// TIA Portal V17 export
// export: Created 2022-07-20T06:59:47.1694326Z, ExportSetting WithDefaults, DisplayName Totally Integrated Automation Portal, DisplayVersion V17, DisplayName TIA Portal Openness, DisplayVersion V17, DisplayName TIA Portal Version Control Interface, DisplayVersion V17, DisplayName SINAMICS Startdrive Advanced, DisplayVersion V17, DisplayName SINAMICS Startdrive G130, G150, S120, S150, SINAMICS MV, S210, DisplayVersion V17, DisplayName SINAMICS Startdrive G110M, G120, G120C, G120D, G120P, G115D, DisplayVersion V17, DisplayName STEP 7 Professional, DisplayVersion V17, DisplayName STEP 7 Safety, DisplayVersion V17, DisplayName WinCC Advanced, DisplayVersion V17
FUNCTION_BLOCK "FB10112_OrientalMotorModbusManager"   // FB10112, LAD
TITLE = FB10112_OrientalMotorModbusManager
{ S7_Optimized_Access := 'TRUE' }
AUTHOR : Anirouddh
FAMILY : 1011x_ORIENTAL_MOTOR
VERSION : 1.0
// Release note : 
// 1.0 - Feature developped
// stored: AutoNumber false, IsIECCheckEnabled false, IsRetainMemResEnabled false, MemoryReserve 100, SetENOAutomatically false, UDAEnableTagReadback false
   VAR_INPUT
      MotorInError : Bool;
      OriginPosition : Real;
      WaitingPosition : Real;
      WorkingPosition : Real;
      StepsMmRatio : Real := 500.0;
      RequestAcknowledge : Bool;
      RequestHoming : Bool;
      RequestGoToOriginPosition : Bool;
      RequestGoToWaitingPosition : Bool;
      RequestGoToWorkingPosition : Bool;
      RequestReadActualPosition : Bool;
      RequestReadOriginPosition : Bool;
      RequestReadWaitingPosition : Bool;
      RequestReadWorkingPosition : Bool;
      RequestWriteOriginPosition : Bool;
      RequestWriteWaitingPosition : Bool;
      RequestWriteWorkingPosition : Bool;
      ModbusRequestDone : Bool;
      ModbusDataRegisterToReceive_0 : Int;
      ModbusDataRegisterToReceive_1 : Int;
   END_VAR
   VAR_OUTPUT
      OrientalMotorOutputCommands : "stOrientalModbusStepperMotorCommandOutputs";
      ActualPosition : Real;
      ActualOriginPosition : Real;
      ActualWaitingPosition : Real;
      ActualWorkingPosition : Real;
      HomingDone : Bool;
      IsInOriginPosition : Bool;
      IsInWaitingPosition : Bool;
      IsInWorkingPosition : Bool;
      ReadActualPositionDone : Bool;
      ReadOriginPositionDone : Bool;
      ReadWaitingPositionDone : Bool;
      ReadWorkingPositionDone : Bool;
      ReadAlarmCodeDone : Bool;
      WriteOriginPositionDone : Bool;
      WriteWaitingPositionDone : Bool;
      WriteWorkingPositionDone : Bool;
      StartModbusRtuCommunication : Bool;
      ModbusRtuDataAddress : UInt;
      ModbusRtuDataLength : UInt;
      ModbusRtuMode : USInt;
      ModbusDataRegisterToSend_0 : Int;
      ModbusDataRegisterToSend_1 : Int;
      AlarmStatus : DInt;
      MaterialOK : Bool;
   END_VAR
   VAR
      RequestMotorStartUp : Bool;
      MotorStartUpStateDiagram : Int;
      ModbusCommunicationStateDiagram : Int;
      MotorMovementStateDiagram : Int;
      MotorAlarmManagementStateDiagram : Int;
      ResetStructure : Array[0..31] of Bool;
      R_TRIG_ModbusRequestDone { S7_SetPoint := 'True'} : R_TRIG;
      R_TRIG_RequestHoming { S7_SetPoint := 'True'} : R_TRIG;
      R_TRIG_RequestGoToOriginPosition { S7_SetPoint := 'True'} : R_TRIG;
      R_TRIG_RequestGoToWaitingPosition { S7_SetPoint := 'True'} : R_TRIG;
      R_TRIG_RequestGoToWorkingPosition { S7_SetPoint := 'True'} : R_TRIG;
      R_TRIG_RequestAcknowledge { S7_SetPoint := 'True'} : R_TRIG;
      F_TRIG_MotorInError { S7_SetPoint := 'True'} : F_TRIG;
      TON_HomingSignal { S7_SetPoint := 'True'} : TON_TIME;
      TON_GoToOriginPositionSignal { S7_SetPoint := 'True'} : TON_TIME;
      TON_GoToWaitingPositionSignal { S7_SetPoint := 'True'} : TON_TIME;
      TON_GoToWorkingPositionSignal { S7_SetPoint := 'True'} : TON_TIME;
      TON_AlarmResetSignal { S7_SetPoint := 'True'} : TON_TIME;
   END_VAR
   VAR_TEMP
      ActualPositionTemp : DInt;
      ActualOriginPositionTemp : DInt;
      ActualWaitingPositionTemp : DInt;
      ActualWorkingPositionTemp : DInt;
      ErrorCodeTemp : DInt;
   END_VAR
   VAR CONSTANT
      WAIT_FOR_MOTOR_START_UP : Int := 0;
      INITIALIZE_ORIGIN_POSITION : Int := 10;
      INITIALIZE_WAITING_POSITION : Int := 20;
      INITIALIZE_WORKING_POSITION : Int := 30;
      MOTOR_START_UP_DONE : Int := 40;
      "==========" : Bool;
      WAIT_FOR_MODBUS_COMMUNICATION_REQUEST : Int := 0;
      READ_ACTUAL_POSITION : Int := 10;
      READ_ORIGIN_POSITION : Int := 20;
      READ_WAITING_POSITION : Int := 30;
      READ_WORKING_POSITION : Int := 40;
      WRITE_ORIGIN_POSITION : Int := 50;
      WRITE_WAITING_POSITION : Int := 60;
      WRITE_WORKING_POSITION : Int := 70;
      MODBUS_COMMUNICATION_DONE : Int := 80;
      "==========_1" : Bool;
      WAIT_FOR_MOVEMENT_REQUEST : Int := 0;
      HOMING : Int := 10;
      GO_TO_ORIGIN_POSITION : Int := 20;
      GO_TO_WAITING_POSITION : Int := 30;
      GO_TO_WORKING_POSITION : Int := 40;
      MOVEMENT_DONE : Int := 50;
      "==========_2" : Bool;
      WAIT_FOR_MOTOR_ERROR : Int := 0;
      RESET_MOTOR_COMMUNICATION_MOVEMENT : Int := 10;
      ALARM_RESET : Int := 20;
      GATHER_ERROR_CODE : Int := 30;
      MOTOR_ERROR_MANAGEMENT_DONE : Int := 40;
   END_VAR
BEGIN

REGION Network 1 (SCL): First Scan
   IF "FirstScan" THEN
       #RequestMotorStartUp := TRUE;
       #HomingDone := TRUE;
       #IsInOriginPosition := FALSE;
       #IsInWaitingPosition := FALSE;
       #IsInWorkingPosition := FALSE;
       #ReadActualPositionDone := FALSE;
       #ReadOriginPositionDone := FALSE;
       #ReadWaitingPositionDone := FALSE;
       #ReadWorkingPositionDone := FALSE;
       #ReadAlarmCodeDone := FALSE;
       #WriteOriginPositionDone := FALSE;
       #WriteWaitingPositionDone := FALSE;
       #WriteWorkingPositionDone := FALSE;
       #OrientalMotorOutputCommands.Start := FALSE;
       #OrientalMotorOutputCommands.Stop := FALSE;
       #OrientalMotorOutputCommands.AlarmReset := FALSE;
       #OrientalMotorOutputCommands.M0 := FALSE;
       #OrientalMotorOutputCommands.M1 := FALSE;
       #OrientalMotorOutputCommands.M2 := FALSE;
       #ModbusCommunicationStateDiagram := #WAIT_FOR_MODBUS_COMMUNICATION_REQUEST;
       #MotorMovementStateDiagram := #WAIT_FOR_MOVEMENT_REQUEST;
       #MaterialOK := FALSE;
   END_IF;
END_REGION

REGION Network 2 (SCL): Edge Signals and Timers
   REGION EGDE SIGNALS
       #R_TRIG_ModbusRequestDone(CLK := #ModbusRequestDone AND
                                 (#MotorStartUpStateDiagram = #INITIALIZE_ORIGIN_POSITION OR
                                 #MotorStartUpStateDiagram = #INITIALIZE_WAITING_POSITION OR
                                 #MotorStartUpStateDiagram = #INITIALIZE_WORKING_POSITION));
       #R_TRIG_RequestHoming(CLK := #MotorMovementStateDiagram = #WAIT_FOR_MOVEMENT_REQUEST AND #RequestHoming);
       #R_TRIG_RequestGoToOriginPosition(CLK := #MotorMovementStateDiagram = #WAIT_FOR_MOVEMENT_REQUEST AND #RequestGoToOriginPosition);
       #R_TRIG_RequestGoToWaitingPosition(CLK := #MotorMovementStateDiagram = #WAIT_FOR_MOVEMENT_REQUEST AND #RequestGoToWaitingPosition);
       #R_TRIG_RequestGoToWorkingPosition(CLK := #MotorMovementStateDiagram = #WAIT_FOR_MOVEMENT_REQUEST AND #RequestGoToWorkingPosition);
       #F_TRIG_MotorInError(CLK := #MotorAlarmManagementStateDiagram = #WAIT_FOR_MOTOR_ERROR AND #MotorInError);
       #R_TRIG_RequestAcknowledge(CLK := #MotorAlarmManagementStateDiagram = #WAIT_FOR_MOTOR_ERROR AND #RequestAcknowledge);
   END_REGION


   REGION TIMERS
       //HomingSignal
       #TON_HomingSignal(IN := #MotorMovementStateDiagram = #HOMING,
                         PT := T#15s);

       //GoToOriginPositionSiganl
       #TON_GoToOriginPositionSignal(IN := #MotorMovementStateDiagram = #GO_TO_ORIGIN_POSITION,
                                     PT := T#200ms);

       //GoToWaitingPositionSignal
       #TON_GoToWaitingPositionSignal(IN := #MotorMovementStateDiagram = #GO_TO_WAITING_POSITION,
                                      PT := T#200ms);

       //GoToWorkingPositionSignal
       #TON_GoToWorkingPositionSignal(IN := #MotorMovementStateDiagram = #GO_TO_WORKING_POSITION,
                                      PT := T#200ms);

       //AlarmResetSignal
       #TON_AlarmResetSignal(IN := #MotorAlarmManagementStateDiagram = #ALARM_RESET,
                             PT := T#500ms);
   END_REGION
END_REGION

REGION Network 3 (SCL): Motor Start Up Management
   CASE #MotorStartUpStateDiagram OF
       #WAIT_FOR_MOTOR_START_UP:
           IF #RequestMotorStartUp AND #RequestAcknowledge THEN
               #MotorStartUpStateDiagram := #INITIALIZE_ORIGIN_POSITION;
           END_IF;
       #INITIALIZE_ORIGIN_POSITION:
           #StartModbusRtuCommunication := TRUE;
           #ModbusRtuDataAddress := 41025;
           #ModbusRtuDataLength := 2;
           #ModbusRtuMode := "MODBUS_RTU_WRITE_MODE";
           "FC10332_DWordTo2Words"(DWord_Input := REAL_TO_DINT(#OriginPosition * #StepsMmRatio),
                                Word_HighWeight => #ModbusDataRegisterToSend_0,
                                Word_LowWeight => #ModbusDataRegisterToSend_1);
           IF #R_TRIG_ModbusRequestDone.Q THEN
               #StartModbusRtuCommunication := FALSE;
               #MotorStartUpStateDiagram := #INITIALIZE_WAITING_POSITION;
           END_IF;
       #INITIALIZE_WAITING_POSITION:
           #StartModbusRtuCommunication := TRUE;
           #ModbusRtuDataAddress := 41027;
           #ModbusRtuDataLength := 2;
           #ModbusRtuMode := "MODBUS_RTU_WRITE_MODE";
           "FC10332_DWordTo2Words"(DWord_Input := REAL_TO_DINT(#WaitingPosition * #StepsMmRatio),
                                Word_HighWeight => #ModbusDataRegisterToSend_0,
                                Word_LowWeight => #ModbusDataRegisterToSend_1);
           IF #R_TRIG_ModbusRequestDone.Q THEN
               #StartModbusRtuCommunication := FALSE;
               #MotorStartUpStateDiagram := #INITIALIZE_WORKING_POSITION;
           END_IF;
       #INITIALIZE_WORKING_POSITION:
           #StartModbusRtuCommunication := TRUE;
           #ModbusRtuDataAddress := 40063;
           #ModbusRtuDataLength := 2;
           #ModbusRtuMode := "MODBUS_RTU_WRITE_MODE";
           "FC10332_DWordTo2Words"(DWord_Input := REAL_TO_DINT(#WorkingPosition * #StepsMmRatio),
                                Word_HighWeight => #ModbusDataRegisterToSend_0,
                                Word_LowWeight => #ModbusDataRegisterToSend_1);
           IF #R_TRIG_ModbusRequestDone.Q THEN
               #StartModbusRtuCommunication := FALSE;
               #MotorStartUpStateDiagram := #MOTOR_START_UP_DONE;
           END_IF;
       #MOTOR_START_UP_DONE:
           #MaterialOK := TRUE;
           #RequestMotorStartUp := FALSE;
   END_CASE;
END_REGION

REGION Network 4 (SCL): Modbus Communication Management
   CASE #ModbusCommunicationStateDiagram OF
       #WAIT_FOR_MODBUS_COMMUNICATION_REQUEST:
           IF #RequestReadActualPosition THEN
               #ReadActualPositionDone := FALSE;
               #ReadOriginPositionDone := FALSE;
               #ReadWaitingPositionDone := FALSE;
               #ReadWorkingPositionDone := FALSE;
               #WriteOriginPositionDone := FALSE;
               #WriteWaitingPositionDone := FALSE;
               #WriteWorkingPositionDone := FALSE;
               #ModbusCommunicationStateDiagram := #READ_ACTUAL_POSITION;
           ELSIF #RequestReadOriginPosition THEN
               #ReadActualPositionDone := FALSE;
               #ReadOriginPositionDone := FALSE;
               #ReadWaitingPositionDone := FALSE;
               #ReadWorkingPositionDone := FALSE;
               #WriteOriginPositionDone := FALSE;
               #WriteWaitingPositionDone := FALSE;
               #WriteWorkingPositionDone := FALSE;
               #ModbusCommunicationStateDiagram := #READ_ORIGIN_POSITION;
           ELSIF #RequestReadWaitingPosition THEN
               #ReadActualPositionDone := FALSE;
               #ReadOriginPositionDone := FALSE;
               #ReadWaitingPositionDone := FALSE;
               #ReadWorkingPositionDone := FALSE;
               #WriteOriginPositionDone := FALSE;
               #WriteWaitingPositionDone := FALSE;
               #WriteWorkingPositionDone := FALSE;
               #ModbusCommunicationStateDiagram := #READ_WAITING_POSITION;
           ELSIF #RequestReadWorkingPosition THEN
               #ReadActualPositionDone := FALSE;
               #ReadOriginPositionDone := FALSE;
               #ReadWaitingPositionDone := FALSE;
               #ReadWorkingPositionDone := FALSE;
               #WriteOriginPositionDone := FALSE;
               #WriteWaitingPositionDone := FALSE;
               #WriteWorkingPositionDone := FALSE;
               #ModbusCommunicationStateDiagram := #READ_WORKING_POSITION;
           ELSIF #RequestWriteOriginPosition THEN
               #ReadActualPositionDone := FALSE;
               #ReadOriginPositionDone := FALSE;
               #ReadWaitingPositionDone := FALSE;
               #ReadWorkingPositionDone := FALSE;
               #WriteOriginPositionDone := FALSE;
               #WriteWaitingPositionDone := FALSE;
               #WriteWorkingPositionDone := FALSE;
               #ModbusCommunicationStateDiagram := #WRITE_ORIGIN_POSITION;
           ELSIF #RequestWriteWaitingPosition THEN
               #ReadActualPositionDone := FALSE;
               #ReadOriginPositionDone := FALSE;
               #ReadWaitingPositionDone := FALSE;
               #ReadWorkingPositionDone := FALSE;
               #WriteOriginPositionDone := FALSE;
               #WriteWaitingPositionDone := FALSE;
               #WriteWorkingPositionDone := FALSE;
               #ModbusCommunicationStateDiagram := #WRITE_WAITING_POSITION;
           ELSIF #RequestWriteWorkingPosition THEN
               #ReadActualPositionDone := FALSE;
               #ReadOriginPositionDone := FALSE;
               #ReadWaitingPositionDone := FALSE;
               #ReadWorkingPositionDone := FALSE;
               #WriteOriginPositionDone := FALSE;
               #WriteWaitingPositionDone := FALSE;
               #WriteWorkingPositionDone := FALSE;
               #ModbusCommunicationStateDiagram := #WRITE_WORKING_POSITION;
           END_IF;
       #READ_ACTUAL_POSITION:
           #StartModbusRtuCommunication := TRUE;
           #ModbusRtuDataAddress := 40205;
           #ModbusRtuDataLength := 2;
           #ModbusRtuMode := "MODBUS_RTU_READ_MODE";
           IF #ModbusRequestDone THEN
               "FC10012_2IntToDint"(HighInt := #ModbusDataRegisterToReceive_0,
                                    LowInt := #ModbusDataRegisterToReceive_1,
                                    Output_DInt => #ActualPositionTemp);
               #ActualPosition := DINT_TO_REAL(#ActualPositionTemp) / #StepsMmRatio;
               #ReadActualPositionDone := TRUE;
               #StartModbusRtuCommunication := FALSE;
               #ModbusCommunicationStateDiagram := #MODBUS_COMMUNICATION_DONE;
           END_IF;
       #READ_ORIGIN_POSITION:
           #StartModbusRtuCommunication := TRUE;
           #ModbusRtuDataAddress := 41025;
           #ModbusRtuDataLength := 2;
           #ModbusRtuMode := "MODBUS_RTU_READ_MODE";
           IF #ModbusRequestDone THEN
               "FC10012_2IntToDint"(HighInt := #ModbusDataRegisterToReceive_0,
                                    LowInt := #ModbusDataRegisterToReceive_1,
                                    Output_DInt => #ActualOriginPositionTemp);
               #ActualOriginPosition := DINT_TO_REAL(#ActualOriginPositionTemp) / #StepsMmRatio;
               #ReadOriginPositionDone := TRUE;
               #StartModbusRtuCommunication := FALSE;
               #ModbusCommunicationStateDiagram := #MODBUS_COMMUNICATION_DONE;
           END_IF;
       #READ_WAITING_POSITION:
           #StartModbusRtuCommunication := TRUE;
           #ModbusRtuDataAddress := 41027;
           #ModbusRtuDataLength := 2;
           #ModbusRtuMode := "MODBUS_RTU_READ_MODE";
           IF #ModbusRequestDone THEN
               "FC10012_2IntToDint"(HighInt := #ModbusDataRegisterToReceive_0,
                                    LowInt := #ModbusDataRegisterToReceive_1,
                                    Output_DInt => #ActualWaitingPositionTemp);
               #ActualWaitingPosition := DINT_TO_REAL(#ActualWaitingPositionTemp) / #StepsMmRatio;
               #ReadWaitingPositionDone := TRUE;
               #StartModbusRtuCommunication := FALSE;
               #ModbusCommunicationStateDiagram := #MODBUS_COMMUNICATION_DONE;
           END_IF;
       #READ_WORKING_POSITION:
           #StartModbusRtuCommunication := TRUE;
           #ModbusRtuDataAddress := 41029;
           #ModbusRtuDataLength := 2;
           #ModbusRtuMode := "MODBUS_RTU_READ_MODE";
           IF #ModbusRequestDone THEN
               "FC10012_2IntToDint"(HighInt := #ModbusDataRegisterToReceive_0,
                                    LowInt := #ModbusDataRegisterToReceive_1,
                                    Output_DInt => #ActualWorkingPositionTemp);
               #ActualWorkingPosition := DINT_TO_REAL(#ActualWorkingPositionTemp) / #StepsMmRatio;
               #ReadWorkingPositionDone := TRUE;
               #StartModbusRtuCommunication := FALSE;
               #ModbusCommunicationStateDiagram := #MODBUS_COMMUNICATION_DONE;
           END_IF;
       #WRITE_ORIGIN_POSITION:
           REGION To test later
       (*    #StartModbusRtuCommunication := TRUE;
           #ModbusRtuDataAddress := 44929;
           #ModbusRtuDataLength := 14;
           #ModbusRtuMode := "MODBUS_RTU_WRITE_MODE";
           (*Process Line Update*)
           //Name -> Line Number
           #ModbusDataRegisterToSend[0] := 0;
           #ModbusDataRegisterToSend[1] := 1;
           //Operation Type
           #ModbusDataRegisterToSend[2] := 1; //AbsolutePositionning
           #ModbusDataRegisterToSend[3] := 0;
           //Position
           "FC10011_DintTo2Int"(Dint_Input := REAL_TO_DINT(#OriginPosition * #StepMmRatio),
                                Int_HighWeight => #ModbusDataRegisterToSend[4],
                                Int_LowWeight => #ModbusDataRegisterToSend[5]);
           //Speed
           "FC10011_DintTo2Int"(Dint_Input := 20000,
                                Int_HighWeight => #ModbusDataRegisterToSend[6],
                                Int_LowWeight => #ModbusDataRegisterToSend[7]);
           //Acceleration
           "FC10011_DintTo2Int"(Dint_Input := REAL_TO_DINT(100.0 * 1000.0), //Value * Ratio(for precision)
                                Int_HighWeight => #ModbusDataRegisterToSend[8],
                                Int_LowWeight => #ModbusDataRegisterToSend[9]);
           //Deceleration
           "FC10011_DintTo2Int"(Dint_Input := REAL_TO_DINT(100.0 * 1000.0), //Value * Ratio(for precision)
                                Int_HighWeight => #ModbusDataRegisterToSend[10],
                                Int_LowWeight => #ModbusDataRegisterToSend[11]);
           //Current Limit
           "FC10011_DintTo2Int"(Dint_Input := REAL_TO_DINT(100.0 * 10), //Value * Ratio(for precision)
                                Int_HighWeight => #ModbusDataRegisterToSend[12],
                                Int_LowWeight => #ModbusDataRegisterToSend[13]);
           IF #ModbusRequestDone THEN
               #WriteOriginPositionDone := TRUE;
               #StartModbusRtuCommunication := FALSE;
               #ModbusCommunicationStateDiagram := #MODBUS_COMMUNICATION_DONE;
           END_IF; *)
           END_REGION
           #StartModbusRtuCommunication := TRUE;
           #ModbusRtuDataAddress := 41025;
           #ModbusRtuDataLength := 2;
           #ModbusRtuMode := "MODBUS_RTU_WRITE_MODE";
           "FC10332_DWordTo2Words"(DWord_Input := REAL_TO_DINT(#OriginPosition * #StepsMmRatio),
                                Word_HighWeight => #ModbusDataRegisterToSend_0,
                                Word_LowWeight => #ModbusDataRegisterToSend_1);
           IF #ModbusRequestDone THEN
               #WriteOriginPositionDone := TRUE;
               #StartModbusRtuCommunication := FALSE;
               #ModbusCommunicationStateDiagram := #MODBUS_COMMUNICATION_DONE;
           END_IF;
       #WRITE_WAITING_POSITION:
           REGION To test later
           (*        #StartModbusRtuCommunication := TRUE;
           #ModbusRtuDataAddress := 44943;
           #ModbusRtuDataLength := 14;
           #ModbusRtuMode := "MODBUS_RTU_WRITE_MODE";
           (*Process Line Update*)
           //Name -> Line Number
           #ModbusDataRegisterToSend[0] := 0;
           #ModbusDataRegisterToSend[1] := 2;
           //Operation Type
           #ModbusDataRegisterToSend[2] := 1; //AbsolutePositionning
           #ModbusDataRegisterToSend[3] := 0;
           //Position
           "FC10011_DintTo2Int"(Dint_Input := REAL_TO_DINT(#WaitingPosition * #StepMmRatio),
                                Int_HighWeight => #ModbusDataRegisterToSend[4],
                                Int_LowWeight => #ModbusDataRegisterToSend[5]);
           //Speed
           "FC10011_DintTo2Int"(Dint_Input := 20000,
                                Int_HighWeight => #ModbusDataRegisterToSend[6],
                                Int_LowWeight => #ModbusDataRegisterToSend[7]);
           //Acceleration
           "FC10011_DintTo2Int"(Dint_Input := REAL_TO_DINT(100.0 * 1000.0), //Value * Ratio(for precision)
                                Int_HighWeight => #ModbusDataRegisterToSend[8],
                                Int_LowWeight => #ModbusDataRegisterToSend[9]);
           //Deceleration
           "FC10011_DintTo2Int"(Dint_Input := REAL_TO_DINT(100.0 * 1000.0), //Value * Ratio(for precision)
                                Int_HighWeight => #ModbusDataRegisterToSend[10],
                                Int_LowWeight => #ModbusDataRegisterToSend[11]);
           //Current Limit
           "FC10011_DintTo2Int"(Dint_Input := REAL_TO_DINT(100.0 * 10), //Value * Ratio(for precision)
                                Int_HighWeight => #ModbusDataRegisterToSend[12],
                                Int_LowWeight => #ModbusDataRegisterToSend[13]);
           IF #ModbusRequestDone THEN
               #WriteWaitingPositionDone := TRUE;
               #StartModbusRtuCommunication := FALSE;
               #ModbusCommunicationStateDiagram := #MODBUS_COMMUNICATION_DONE;
           END_IF; *)
           END_REGION
           #StartModbusRtuCommunication := TRUE;
           #ModbusRtuDataAddress := 41027;
           #ModbusRtuDataLength := 2;
           #ModbusRtuMode := "MODBUS_RTU_WRITE_MODE";
           "FC10332_DWordTo2Words"(DWord_Input := REAL_TO_DINT(#WaitingPosition * #StepsMmRatio),
                                Word_HighWeight => #ModbusDataRegisterToSend_0,
                                Word_LowWeight => #ModbusDataRegisterToSend_1);
           IF #ModbusRequestDone THEN
               #WriteWaitingPositionDone := TRUE;
               #StartModbusRtuCommunication := FALSE;
               #ModbusCommunicationStateDiagram := #MODBUS_COMMUNICATION_DONE;
           END_IF;
       #WRITE_WORKING_POSITION:
           REGION To test later
           (*    #StartModbusRtuCommunication := TRUE;
               #ModbusRtuDataAddress := 44957;
               #ModbusRtuDataLength := 14;
               #ModbusRtuMode := "MODBUS_RTU_WRITE_MODE";
           (*Process Line Update*)
               //Name -> Line Number
               #ModbusDataRegisterToSend[0] := 0;
               #ModbusDataRegisterToSend[1] := 3;
               //Operation Type
               #ModbusDataRegisterToSend[2] := 1; //AbsolutePositionning
               #ModbusDataRegisterToSend[3] := 0;
               //Position
               "FC10011_DintTo2Int"(Dint_Input := REAL_TO_DINT(#WorkingPosition * #StepMmRatio),
                                    Int_HighWeight => #ModbusDataRegisterToSend[4],
                                    Int_LowWeight => #ModbusDataRegisterToSend[5]);
               //Speed
               "FC10011_DintTo2Int"(Dint_Input := 20000,
                                    Int_HighWeight => #ModbusDataRegisterToSend[6],
                                    Int_LowWeight => #ModbusDataRegisterToSend[7]);
               //Acceleration
               "FC10011_DintTo2Int"(Dint_Input := REAL_TO_DINT(100.0 * 1000.0), //Value * Ratio(for precision)
                                    Int_HighWeight => #ModbusDataRegisterToSend[8],
                                    Int_LowWeight => #ModbusDataRegisterToSend[9]);
               //Deceleration
               "FC10011_DintTo2Int"(Dint_Input := REAL_TO_DINT(100.0 * 1000.0), //Value * Ratio(for precision)
                                    Int_HighWeight => #ModbusDataRegisterToSend[10],
                                    Int_LowWeight => #ModbusDataRegisterToSend[11]);
               //Current Limit
               "FC10011_DintTo2Int"(Dint_Input := REAL_TO_DINT(100.0 * 10), //Value * Ratio(for precision)
                                    Int_HighWeight => #ModbusDataRegisterToSend[12],
                                    Int_LowWeight => #ModbusDataRegisterToSend[13]);
               IF #ModbusRequestDone THEN
                   #WriteWorkingPositionDone := TRUE;
                   #StartModbusRtuCommunication := FALSE;
                   #ModbusCommunicationStateDiagram := #MODBUS_COMMUNICATION_DONE;

               END_IF; *)
           END_REGION
           #StartModbusRtuCommunication := TRUE;
           #ModbusRtuDataAddress := 41029;
           #ModbusRtuDataLength := 2;
           #ModbusRtuMode := "MODBUS_RTU_WRITE_MODE";
           "FC10332_DWordTo2Words"(DWord_Input := REAL_TO_DINT(#WorkingPosition * #StepsMmRatio),
                                Word_HighWeight => #ModbusDataRegisterToSend_0,
                                Word_LowWeight => #ModbusDataRegisterToSend_1);
           IF #ModbusRequestDone THEN
               #WriteWorkingPositionDone := TRUE;
               #StartModbusRtuCommunication := FALSE;
               #ModbusCommunicationStateDiagram := #MODBUS_COMMUNICATION_DONE;
           END_IF;
       #MODBUS_COMMUNICATION_DONE:
           #ModbusCommunicationStateDiagram := #WAIT_FOR_MODBUS_COMMUNICATION_REQUEST;
   END_CASE;
END_REGION

REGION Network 5 (SCL): Motor Movement Management
   CASE #MotorMovementStateDiagram OF
       #WAIT_FOR_MOVEMENT_REQUEST:
           IF #R_TRIG_RequestHoming.Q THEN
               #HomingDone := FALSE;
               #IsInOriginPosition := FALSE;
               #IsInWaitingPosition := FALSE;
               #IsInWorkingPosition := FALSE;
               #MotorMovementStateDiagram := #HOMING;
           ELSIF #R_TRIG_RequestGoToOriginPosition.Q THEN
               #HomingDone := FALSE;
               #IsInOriginPosition := FALSE;
               #IsInWaitingPosition := FALSE;
               #IsInWorkingPosition := FALSE;
               #MotorMovementStateDiagram := #GO_TO_ORIGIN_POSITION;
           ELSIF #R_TRIG_RequestGoToWaitingPosition.Q THEN
               #HomingDone := FALSE;
               #IsInOriginPosition := FALSE;
               #IsInWaitingPosition := FALSE;
               #IsInWorkingPosition := FALSE;
               #MotorMovementStateDiagram := #GO_TO_WAITING_POSITION;
           ELSIF #R_TRIG_RequestGoToWorkingPosition.Q THEN
               #HomingDone := FALSE;
               #IsInOriginPosition := FALSE;
               #IsInWaitingPosition := FALSE;
               #IsInWorkingPosition := FALSE;
               #MotorMovementStateDiagram := #GO_TO_WORKING_POSITION;
           END_IF;
       #HOMING:
           #OrientalMotorOutputCommands.Start := FALSE;
           #OrientalMotorOutputCommands.M0 := FALSE;
           #OrientalMotorOutputCommands.M1 := FALSE;
           #OrientalMotorOutputCommands.Home := TRUE;
           IF #TON_HomingSignal.Q THEN
               #OrientalMotorOutputCommands.Start := FALSE;
               #OrientalMotorOutputCommands.M0 := FALSE;
               #OrientalMotorOutputCommands.M1 := FALSE;
               #OrientalMotorOutputCommands.Home := FALSE;
               #HomingDone := TRUE;
               RESET_TIMER(#TON_HomingSignal);
               #MotorMovementStateDiagram := #GO_TO_WAITING_POSITION;
           END_IF;
       #GO_TO_ORIGIN_POSITION:
           #OrientalMotorOutputCommands.Start := TRUE;
           #OrientalMotorOutputCommands.M0 := FALSE;
           #OrientalMotorOutputCommands.M1 := FALSE;
           IF #TON_GoToOriginPositionSignal.Q THEN
               #OrientalMotorOutputCommands.Start := FALSE;
               #OrientalMotorOutputCommands.M0 := FALSE;
               #OrientalMotorOutputCommands.M1 := FALSE;
               #IsInOriginPosition := TRUE;
               RESET_TIMER(#TON_GoToOriginPositionSignal);
               #MotorMovementStateDiagram := #MOVEMENT_DONE;
           END_IF;
       #GO_TO_WAITING_POSITION:
           #OrientalMotorOutputCommands.Start := TRUE;
           #OrientalMotorOutputCommands.M0 := TRUE;
           #OrientalMotorOutputCommands.M1 := FALSE;
           IF #TON_GoToWaitingPositionSignal.Q THEN
               #OrientalMotorOutputCommands.Start := FALSE;
               #OrientalMotorOutputCommands.M0 := FALSE;
               #OrientalMotorOutputCommands.M1 := FALSE;
               #IsInWaitingPosition := TRUE;
               RESET_TIMER(#TON_GoToWaitingPositionSignal);
               #MotorMovementStateDiagram := #MOVEMENT_DONE;
           END_IF;
       #GO_TO_WORKING_POSITION:
           #OrientalMotorOutputCommands.Start := TRUE;
           #OrientalMotorOutputCommands.M0 := FALSE;
           #OrientalMotorOutputCommands.M1 :=TRUE;
           IF #TON_GoToWorkingPositionSignal.Q THEN
               #OrientalMotorOutputCommands.Start := FALSE;
               #OrientalMotorOutputCommands.M0 := FALSE;
               #OrientalMotorOutputCommands.M1 := FALSE;
               #IsInWorkingPosition := TRUE;
               RESET_TIMER(#TON_GoToWorkingPositionSignal);
               #MotorMovementStateDiagram := #MOVEMENT_DONE;
           END_IF;
       #MOVEMENT_DONE:
           #MotorMovementStateDiagram := #WAIT_FOR_MOVEMENT_REQUEST;
   END_CASE;
END_REGION

REGION Network 6 (SCL): Motor Error Management
   CASE #MotorAlarmManagementStateDiagram OF
       #WAIT_FOR_MOTOR_ERROR:
           IF #F_TRIG_MotorInError.Q THEN
               #ReadAlarmCodeDone := FALSE;
               #MotorAlarmManagementStateDiagram := #RESET_MOTOR_COMMUNICATION_MOVEMENT;
           ELSIF #R_TRIG_RequestAcknowledge.Q THEN
               #ReadAlarmCodeDone := FALSE;
               #MotorAlarmManagementStateDiagram := #ALARM_RESET;
           END_IF;
       #RESET_MOTOR_COMMUNICATION_MOVEMENT:
           #ModbusCommunicationStateDiagram := #WAIT_FOR_MODBUS_COMMUNICATION_REQUEST;
           #MotorMovementStateDiagram := #WAIT_FOR_MOVEMENT_REQUEST;
           #OrientalMotorOutputCommands.M0 := FALSE;
           #OrientalMotorOutputCommands.M1 := FALSE;
           #OrientalMotorOutputCommands.M2 := FALSE;
           #OrientalMotorOutputCommands.Start := FALSE;
           #OrientalMotorOutputCommands.Stop := FALSE;
           #StartModbusRtuCommunication := FALSE;
           IF (#ModbusCommunicationStateDiagram = #WAIT_FOR_MODBUS_COMMUNICATION_REQUEST) AND (#MotorMovementStateDiagram = #WAIT_FOR_MOVEMENT_REQUEST) AND NOT (#StartModbusRtuCommunication) THEN
               #MotorAlarmManagementStateDiagram := #GATHER_ERROR_CODE;
           END_IF;
       #ALARM_RESET:
           #OrientalMotorOutputCommands.AlarmReset := TRUE;
           IF #TON_AlarmResetSignal.Q THEN
               #OrientalMotorOutputCommands.AlarmReset := FALSE;
               #MotorAlarmManagementStateDiagram := #GATHER_ERROR_CODE;
           END_IF;
       #GATHER_ERROR_CODE:
           #StartModbusRtuCommunication := TRUE;
           #ModbusRtuDataAddress := 40130;
           #ModbusRtuDataLength := 1;
           #ModbusRtuMode := "MODBUS_RTU_READ_MODE";
           IF #ModbusRequestDone THEN
               "FC10012_2IntToDint"(HighInt := #ModbusDataRegisterToReceive_0,
                                    LowInt := #ModbusDataRegisterToReceive_1,
                                    Output_DInt => #AlarmStatus);
               #ReadAlarmCodeDone := FALSE;
               #StartModbusRtuCommunication := FALSE;
               #MotorAlarmManagementStateDiagram := #MOTOR_ERROR_MANAGEMENT_DONE;
           END_IF;
       #MOTOR_ERROR_MANAGEMENT_DONE:
           #MotorAlarmManagementStateDiagram := #WAIT_FOR_MOTOR_ERROR;
   END_CASE;
END_REGION
END_FUNCTION_BLOCK
